# EPICS autosave request: pslApp/Db/PSL_settings.req
file "ADBase_settings.req", P=$(P), R=$(R)
$(P)$(R)CameraName
$(P)$(R)TIFFComment
